// TwinCAT 3 PLC project Logic_Circuit_Exercises
// ProgramVersion: 3.1.4024.0
// libraries:
//   Tc2_Standard, * (Beckhoff Automation GmbH)
//   Tc2_System, * (Beckhoff Automation GmbH)
//   Tc3_Module, * (Beckhoff Automation GmbH)
// project tree:
//   / PlcTask.TcTTO
//   POUs/ ControlPanel.TcPOU, ITF_Control.TcIO, LampControl.TcPOU, MAIN.TcPOU
// real-time tasks:
//   TASK PlcTask: cycle T#10ms, priority 20, ADS port 350

CONFIGURATION Logic_Circuit_Exercises
    RESOURCE PLC ON TwinCAT3
        TASK PlcTask(INTERVAL := T#10ms, PRIORITY := 20);
        PROGRAM MAIN WITH PlcTask : MAIN;
    END_RESOURCE
END_CONFIGURATION

// ---- POUs/ITF_Control.TcIO
INTERFACE ITF_Control

METHOD GetSwitchS10 : BOOL
VAR_INPUT
END_VAR
END_METHOD

END_INTERFACE

// ---- POUs/MAIN.TcPOU
PROGRAM MAIN
VAR
	MachineControl : ControlPanel;
	MachineLamps : LampControl := (Controller := MachineControl);
END_VAR

MachineLamps.Cycle();

END_PROGRAM

// ---- POUs/ControlPanel.TcPOU
FUNCTION_BLOCK ControlPanel IMPLEMENTS ITF_Control
VAR
	SwitchS10 AT%i* : BOOL;
END_VAR

METHOD GetSwitchS10 : BOOL
VAR_INPUT
END_VAR
GetSwitchS10 := SwitchS10;
END_METHOD

END_FUNCTION_BLOCK

// ---- POUs/LampControl.TcPOU
FUNCTION_BLOCK LampControl
VAR
	LampP1 AT%Q* : BOOL;
	_Control : ITF_Control;
END_VAR

PROPERTY Controller : ITF_Control
GET
Controller := _Control;
END_GET
SET
_Control := Controller;
END_SET
END_PROPERTY

METHOD Cycle : BOOL
VAR_INPUT
END_VAR
LampP1 := _Control.GetSwitchS10();
END_METHOD

END_FUNCTION_BLOCK
